FUNCTION_BLOCK T_ModuleCollectionSetSubModuleInfoStateSuccess EXTENDS T_UnitTestBase
VAR
  list : T_SubModuleCollection(10);
  newModule, newModule2 : T_SubModuleMock; 
  actual1, actual2, result : BOOL;

  PMLSubModuleInfo  : ARRAY[1..10] OF ST_PMLSubUnitInfo;
END_VAR

// Arrange
list.AddModule(newModule);
list.AddModule(newModule2);

//Act
newModule._Currentstate := Tc3_PackML_V2.E_PMLState.ePMLState_Clearing;
newModule2._Currentstate := Tc3_PackML_V2.E_PMLState.ePMLState_Held;

list.SetSubModuleInfoState(PMLSubModuleInfo);

//Assert
actual1:=  PMLSubModuleInfo[1].eState = Tc3_PackML_V2.E_PMLState.ePMLState_Clearing;
actual2:=  PMLSubModuleInfo[2].eState = Tc3_PackML_V2.E_PMLState.ePMLState_Held;

assertion.AssertEquals_BOOL(TRUE, actual1, 'PMLSubModuleInfo[1].eState = Tc3_PackML_V2.E_PMLState.ePMLState_Clearing');
assertion.AssertEquals_BOOL(TRUE, actual2, ' PMLSubModuleInfo[2].eState = Tc3_PackML_V2.E_PMLState.ePMLState_Held');
TestFinished();

END_FUNCTION_BLOCK

(* stored: Version 1.1.0.1, ProductVersion 3.1.4024.12
   POU T_ModuleCollectionSetSubModuleInfoStateSuccess: Id {fd5cc682-4a1e-4e95-b66a-239dad0ae652}, SpecialFunc None *)
